FUNCTION_BLOCK FB_DobraValor
VAR_INPUT
END_VAR
VAR_OUTPUT
END_VAR
VAR
END_VAR

END_FUNCTION_BLOCK

(* stored: Version 1.1.0.1, ProductVersion 3.1.4024.12
   POU FB_DobraValor: Id {a0d78fc3-7bd3-4ddb-8b8d-f042e4984c9b}, SpecialFunc None *)
